// TIA Portal V19 export
TYPE "Positioning_EPOS_Machine_Config"
// stored: Access Published
   STRUCT
      SLS_Vel : LReal;
      DelayMissingCondition : Time;
      Ax : Struct
         LeadScrewPitchVal : LReal;
         MotorRevolution : LReal;
         LoadRevolution : LReal;
         PowerOffDelay : Time;
         MaxRPM_S120_P2000 : LReal;   // inserire il valore esattamente come nel parametro = in RPM
         MaxVel_S120_P2571 : LReal;   // [1000 LU/min] (= Engineering unit) e.g. 1000 = 1000 mm/min
         MaxAcc_S120_P2572 : LReal;   // [1000 LU/s²] (= Engineering unit) e.g. 1000 = 1000 mm/s²
         MaxDec_S120_P2573 : LReal;   // [1000 LU/s²] (= Engineering unit) e.g. 1000 = 1000 mm/s²
         Modulo_S120_P2566 : LReal;   // Inserire Parametro /1000 perchè [LU] (= Engineering unit * 1000) e.g 1000_000 = 1000 mm
         SwLimMinus_S120_P2580 : LReal;   // Inserire Parametro /1000 perchè [LU] (= Engineering unit * 1000) e.g 1000_000 = 1000 mm
         SwLimPlus_S120_P2581 : LReal;   // [Inserire Parametro /1000 perchè LU] (= Engineering unit * 1000) e.g 1000_000 = 1000 mm
      END_STRUCT;
      Fan : Struct
         Presence : Bool;
         DelayOff : Time;
      END_STRUCT;
      Brake_Presence : Bool;
   END_STRUCT;
END_TYPE
